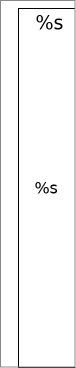
VISUALIZATION Obj_Terminal  // 76x368
VAR_INPUT
	sIndex : STRING;
	sModule : STRING;
	bOffline : BOOL;	
END_VAR
    Rectangle (18,8 57x360), "%s", text variable: sIndex, colour toggle: bOffline
    Rectangle (23,9 53x28), "%s", text variable: sModule
END_VISUALIZATION

(* stored: Version 1.1.0.1, ProductVersion 3.1.4024.12
   Visu Obj_Terminal: Id {86ff6a89-1c50-4749-8443-ce69114b6b44} *)
